{attribute 'GeneratedUsingTerminal: AT2040-0250-0024'}
{attribute addProperty BoxType "AT2040-0250-0024"}
{attribute addProperty Id "A_0105_AT2026_5250_0018_AT2026_5250AT2026_33A3DF1B80"}
{attribute addProperty CRC "928602346"}
{attribute addProperty Size "80"}
TYPE A_0039_AT2040_0250_0024_375958EA EXTENDS AT2040_2EA6C9BF :
STRUCT
	{attribute addProperty Name "A_0105(AT2026-5250-0018) (AT2026-5250)"}
	{attribute addProperty PreviousPort "A_0039(AT2040-0250-0024) : B"}
	A_0105_AT2026_5250_0018_AT2026_5250 : AT2026_33A3DF1B;
END_STRUCT
END_TYPE

(* stored: Version 1.2.0.0, ProductVersion 3.1.4024.9
   DUT A_0039_AT2040_0250_0024_375958EA: Id {a993a8af-83c5-40c8-8ea8-14d0537cfa65} *)
